Universal Robots PolyScope program: Collaboration_CollaborativeAssembly.urp

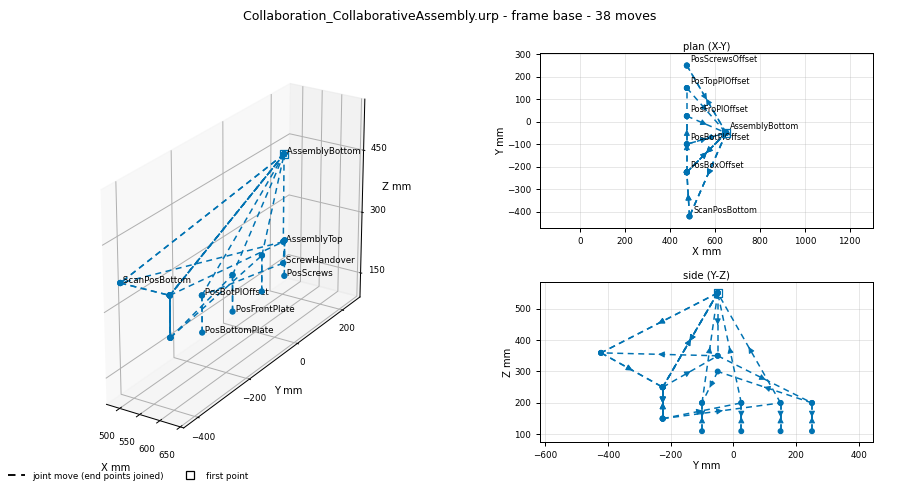
[picture p0: tool path of Collaboration_CollaborativeAssembly.urp in frame base, 38 of 38 moves have a stored position in this frame; points joined in program order, loops and branches not executed]
Program Collaboration_CollaborativeAssembly (installation=Collaboration_CollaborativeAssembly directory=/home/cobot/ursim-5.11.5.1010327/programs createdIn=5.11.5.1010327 lastSavedIn=5.11.5.1010327 robotSerialNumber=20195599999)
Calibrated DH parameters: a=[0, -0.425, -0.3922, 0, 0, 0]; d=[0.1625, 0, 0, 0.1333, 0.0997, 0.0996]; alpha=[1.570796, 0, 0, 1.570796, -1.570796, 0]; deltaTheta=[0, 0, 0, 0, 0, 0]
InitVariablesNode variables(variable(name=qualityCheck, expression=0))
Robot Program (runOnlyOnce=false)
  Wait DigitalInput pin=ib64; digitalValue=1
  Switch expression=GP_int_in[24]
    Case (caseValue=0)
      'Just to start the program in home position'
      SafeHome (positionOptionType=SPEED_AND_ACCELERATION speed=1.047198 acceleration=1.396263 nextMotionTime=2)
    Case (caseValue=1)
      'Keep holding box in place for assembly'
      Switch expression=qualityCheck
        Case (caseValue=1)
          MoveJ speed 60 deg/s, acceleration 80 deg/s^2 (useActiveTCP=true) feature=Workspace1
            Waypoint AssemblyBottom: TCP in base x=650 y=-50 z=550 mm, rx=-1.9651 ry=1.9495 rz=-0.4189 rad; joints [7.029, -130.786, -72.869, -40.345, 268.812, -6.299] deg; TCP offset x=0 y=0 z=100 mm, rx=0 ry=3.1416 rz=0 rad; feature pose in base x=400 y=-300 z=100 mm, rx=0 ry=0 rz=0 rad
        Case (caseValue=2)
          MoveJ speed 60 deg/s, acceleration 80 deg/s^2 (useActiveTCP=true) feature=Workspace1
            Waypoint AssemblyFront: TCP in base x=650 y=-50 z=550 mm, rx=1.5296 ry=-1.5609 rz=-0.9866 rad; joints [11.102, -92.477, -92.844, -147.831, 281.832, -4.972] deg
        Case (caseValue=3)
          MoveJ speed 60 deg/s, acceleration 80 deg/s^2 (useActiveTCP=true) feature=Workspace1
            Waypoint AssemblyTop: TCP in base x=650 y=-50 z=350 mm, rx=0.4964 ry=-0.5461 rz=-1.5185 rad; joints [9.895, -118.031, -57.592, -236.953, 277.963, 7.867] deg
      qualityCheck := 0
    Case (caseValue=2)
      'Pick and hand over box of screws'
      MoveJ speed 60 deg/s, acceleration 80 deg/s^2 (useActiveTCP=true) feature=Workspace1
        Waypoint PosScrewsOffset: motionParameters(blendRadius=0.05); TCP in base x=475 y=250 z=200 mm, rx=1.1931 ry=-1.2328 rz=-1.2341 rad; joints [63.7, -100.587, -125.054, -134.467, 335.594, 0.116] deg
        Waypoint PosScrews: TCP in base x=475 y=250 z=110 mm, rx=1.1931 ry=-1.2328 rz=-1.2341 rad; joints [63.7, -112.802, -128.624, -118.681, 335.594, 0.116] deg
      Wait Sleep waitTime=2
      MoveJ speed 60 deg/s, acceleration 80 deg/s^2 (useActiveTCP=true) feature=Workspace1
        Waypoint PosScrewsOffset: motionParameters(blendRadius=0.05); TCP in base x=475 y=250 z=200 mm, rx=1.1931 ry=-1.2328 rz=-1.2341 rad; joints [63.7, -100.587, -125.054, -134.467, 335.594, 0.116] deg
        Waypoint ScrewHandover: TCP in base x=650 y=-50 z=300 mm, rx=1.1931 ry=-1.2328 rz=-1.2341 rad; joints [11.626, -101.37, -105.835, -152.841, 283.52, 0.028] deg
    Case (caseValue=3)
      'Pick and hand over bottom plate'
      MoveJ speed 60 deg/s, acceleration 80 deg/s^2 (useActiveTCP=true) feature=Workspace1
        Waypoint PosBotPlOffset: motionParameters(blendRadius=0.05); TCP in base x=475 y=-100 z=200 mm, rx=1.1931 ry=-1.2328 rz=-1.2341 rad; joints [8.545, -88.916, -138.241, -132.888, 280.439, 0.026] deg
        Waypoint PosBottomPlate: TCP in base x=475 y=-100 z=110 mm, rx=1.1931 ry=-1.2328 rz=-1.2341 rad; joints [8.545, -105.047, -142.733, -112.265, 280.439, 0.026] deg
      Wait Sleep waitTime=2
      MoveJ speed 60 deg/s, acceleration 80 deg/s^2 (useActiveTCP=true) feature=Workspace1
        Waypoint PosBotPlOffset: motionParameters(blendRadius=0.05); TCP in base x=475 y=-100 z=200 mm, rx=1.1931 ry=-1.2328 rz=-1.2341 rad; joints [8.545, -88.916, -138.241, -132.888, 280.439, 0.026] deg
        Waypoint PlateHandover: TCP in base x=650 y=-50 z=550 mm, rx=1.1931 ry=-1.2328 rz=-1.2341 rad; joints [11.626, -96.186, -74.3, -189.56, 283.52, 0.028] deg
    Case (caseValue=4)
      'Grab and hold box in place for assembly (bottom plate)'
      MoveJ speed 60 deg/s, acceleration 80 deg/s^2 (useActiveTCP=true) feature=Workspace1
        Waypoint PosBoxOffset: motionParameters(blendRadius=0.025); TCP in base x=475 y=-225 z=250 mm, rx=1.1931 ry=-1.2328 rz=-1.2341 rad; joints [-16.123, -91.786, -125.472, -142.788, 255.771, 0.006] deg
        Waypoint PosBox: TCP in base x=475 y=-225 z=149.999 mm, rx=1.1931 ry=-1.2328 rz=-1.2341 rad; joints [-16.123, -104.312, -131.507, -124.226, 255.771, 0.006] deg
      Wait Sleep waitTime=2
      MoveJ speed 60 deg/s, acceleration 80 deg/s^2 (useActiveTCP=true) feature=Workspace1
        Waypoint PosBoxOffset: motionParameters(blendRadius=0.05); TCP in base x=475 y=-225 z=250 mm, rx=1.1931 ry=-1.2328 rz=-1.2341 rad; joints [-16.123, -91.786, -125.472, -142.788, 255.771, 0.006] deg
        Waypoint AssemblyBottom: TCP in base x=650 y=-50 z=550 mm, rx=-1.9651 ry=1.9495 rz=-0.4189 rad; joints [7.029, -130.786, -72.869, -40.345, 268.812, -6.299] deg
    Case (caseValue=5)
      'Check quality of assembly (bottom plate)'
      qualityCheck := 1
      MoveJ speed 60 deg/s, acceleration 80 deg/s^2 (useActiveTCP=true) feature=Workspace1
        Waypoint ScanPosBottom: TCP in base x=486.827 y=-421.362 z=359.312 mm, rx=-0.9579 ry=1.4438 rz=1.2517 rad; joints [-9.744, -105.127, -103.748, -76.262, 359.415, 1.851] deg
    Case (caseValue=6)
      'Put box aside and pick and hand over front plate'
      MoveJ speed 60 deg/s, acceleration 80 deg/s^2 (useActiveTCP=true) feature=Workspace1
        Waypoint PosBoxOffset: motionParameters(blendRadius=0.025); TCP in base x=475 y=-225 z=250 mm, rx=1.1931 ry=-1.2328 rz=-1.2341 rad; joints [-16.123, -91.786, -125.472, -142.788, 255.771, 0.006] deg
        Waypoint PosBox: TCP in base x=475 y=-225 z=149.999 mm, rx=1.1931 ry=-1.2328 rz=-1.2341 rad; joints [-16.123, -104.312, -131.507, -124.226, 255.771, 0.006] deg
      Wait Sleep waitTime=2
      MoveJ speed 60 deg/s, acceleration 80 deg/s^2 (useActiveTCP=true) feature=Workspace1
        Waypoint PosFroPlOffset: motionParameters(blendRadius=0.05); TCP in base x=475 y=25 z=200 mm, rx=1.1931 ry=-1.2328 rz=-1.2341 rad; joints [35.273, -86.753, -140.274, -133.029, 307.167, 0.051] deg
        Waypoint PosFrontPlate: TCP in base x=475 y=25 z=110 mm, rx=1.1931 ry=-1.2328 rz=-1.2341 rad; joints [35.273, -103.744, -144.982, -111.329, 307.167, 0.051] deg
      Wait Sleep waitTime=2
      MoveJ speed 60 deg/s, acceleration 80 deg/s^2 (useActiveTCP=true) feature=Workspace1
        Waypoint PosFroPlOffset: TCP in base x=475 y=25 z=200 mm, rx=1.1931 ry=-1.2328 rz=-1.2341 rad; joints [35.273, -86.753, -140.274, -133.029, 307.167, 0.051] deg
        Waypoint PlateHandover: TCP in base x=650 y=-50 z=550 mm, rx=1.1931 ry=-1.2328 rz=-1.2341 rad; joints [11.626, -96.186, -74.3, -189.56, 283.52, 0.028] deg
    Case (caseValue=7)
      'Grab and hold box in place for assembly (front plate)'
      MoveJ speed 60 deg/s, acceleration 80 deg/s^2 (useActiveTCP=true) feature=Workspace1
        Waypoint PosBoxOffset: motionParameters(blendRadius=0.025); TCP in base x=475 y=-225 z=250 mm, rx=1.1931 ry=-1.2328 rz=-1.2341 rad; joints [-16.123, -91.786, -125.472, -142.788, 255.771, 0.006] deg
        Waypoint PosBox: TCP in base x=475 y=-225 z=149.999 mm, rx=1.1931 ry=-1.2328 rz=-1.2341 rad; joints [-16.123, -104.312, -131.507, -124.226, 255.771, 0.006] deg
      Wait Sleep waitTime=2
      MoveJ speed 60 deg/s, acceleration 80 deg/s^2 (useActiveTCP=true) feature=Workspace1
        Waypoint PosBoxOffset: motionParameters(blendRadius=0.05); TCP in base x=475 y=-225 z=250 mm, rx=1.1931 ry=-1.2328 rz=-1.2341 rad; joints [-16.123, -91.786, -125.472, -142.788, 255.771, 0.006] deg
        Waypoint AssemblyFront: TCP in base x=650 y=-50 z=550 mm, rx=1.5296 ry=-1.5609 rz=-0.9866 rad; joints [11.102, -92.477, -92.844, -147.831, 281.832, -4.972] deg
    Case (caseValue=8)
      'Check quality of assembly (front plate)'
      qualityCheck := 2
      MoveJ speed 60 deg/s, acceleration 80 deg/s^2 (useActiveTCP=true) feature=Workspace1
        Waypoint ScanPosFront: TCP in base x=486.827 y=-421.362 z=359.312 mm, rx=0.0343 ry=2.0931 rz=2.0493 rad; joints [-9.744, -105.127, -103.748, -76.262, 359.415, -67.15] deg
    Case (caseValue=9)
      'Put box aside and pick and hand over top plate'
      MoveJ speed 60 deg/s, acceleration 80 deg/s^2 (useActiveTCP=true) feature=Workspace1
        Waypoint PosBoxOffset: motionParameters(blendRadius=0.025); TCP in base x=475 y=-225 z=250 mm, rx=1.1931 ry=-1.2328 rz=-1.2341 rad; joints [-16.123, -91.786, -125.472, -142.788, 255.771, 0.006] deg
        Waypoint PosBox: TCP in base x=475 y=-225 z=149.999 mm, rx=1.1931 ry=-1.2328 rz=-1.2341 rad; joints [-16.123, -104.312, -131.507, -124.226, 255.771, 0.006] deg
      Wait Sleep waitTime=2
      MoveJ speed 60 deg/s, acceleration 80 deg/s^2 (useActiveTCP=true) feature=Workspace1
        Waypoint PosTopPlOffset: motionParameters(blendRadius=0.05); TCP in base x=475 y=150 z=200 mm, rx=1.1931 ry=-1.2328 rz=-1.2341 rad; joints [54.488, -92.765, -134.302, -133.013, 326.383, 0.084] deg
        Waypoint PosTopPlate: TCP in base x=475 y=150 z=110 mm, rx=1.1931 ry=-1.2328 rz=-1.2341 rad; joints [54.488, -107.468, -138.444, -114.168, 326.383, 0.084] deg
      Wait Sleep waitTime=2
      MoveJ speed 60 deg/s, acceleration 80 deg/s^2 (useActiveTCP=true) feature=Workspace1
        Waypoint PosTopPlOffset: TCP in base x=475 y=150 z=200 mm, rx=1.1931 ry=-1.2328 rz=-1.2341 rad; joints [54.488, -92.765, -134.302, -133.013, 326.383, 0.084] deg
        Waypoint PlateHandover: TCP in base x=650 y=-50 z=550 mm, rx=1.1931 ry=-1.2328 rz=-1.2341 rad; joints [11.626, -96.186, -74.3, -189.56, 283.52, 0.028] deg
    Case (caseValue=10)
      'Grab and hold box in place for assembly (top plate)'
      MoveJ speed 60 deg/s, acceleration 80 deg/s^2 (useActiveTCP=true) feature=Workspace1
        Waypoint PosBoxOffset: motionParameters(blendRadius=0.025); TCP in base x=475 y=-225 z=250 mm, rx=1.1931 ry=-1.2328 rz=-1.2341 rad; joints [-16.123, -91.786, -125.472, -142.788, 255.771, 0.006] deg
        Waypoint PosBox: TCP in base x=475 y=-225 z=149.999 mm, rx=1.1931 ry=-1.2328 rz=-1.2341 rad; joints [-16.123, -104.312, -131.507, -124.226, 255.771, 0.006] deg
      Wait Sleep waitTime=2
      MoveJ speed 60 deg/s, acceleration 80 deg/s^2 (useActiveTCP=true) feature=Workspace1
        Waypoint PosBoxOffset: motionParameters(blendRadius=0.05); TCP in base x=475 y=-225 z=250 mm, rx=1.1931 ry=-1.2328 rz=-1.2341 rad; joints [-16.123, -91.786, -125.472, -142.788, 255.771, 0.006] deg
        Waypoint AssemblyTop: TCP in base x=650 y=-50 z=350 mm, rx=0.4964 ry=-0.5461 rz=-1.5185 rad; joints [9.895, -118.031, -57.592, -236.953, 277.963, 7.867] deg
    Case (caseValue=11)
      'Check quality of assembly (top plate)'
      qualityCheck := 3
      MoveJ speed 60 deg/s, acceleration 80 deg/s^2 (useActiveTCP=true) feature=Workspace1
        Waypoint ScanPosTop: TCP in base x=486.827 y=-421.362 z=359.312 mm, rx=-1.3653 ry=-1.0786 rz=-1.2783 rad; joints [-9.744, -105.127, -103.748, -76.262, 359.415, -168.655] deg
    Case (caseValue=2147483647)
      'Do nothing (just handshake)'
  Set DigitalOutput pin=ob64; digitalValue=1
  Wait DigitalInput pin=ib64; digitalValue=0
  Set DigitalOutput pin=ob64; digitalValue=0
